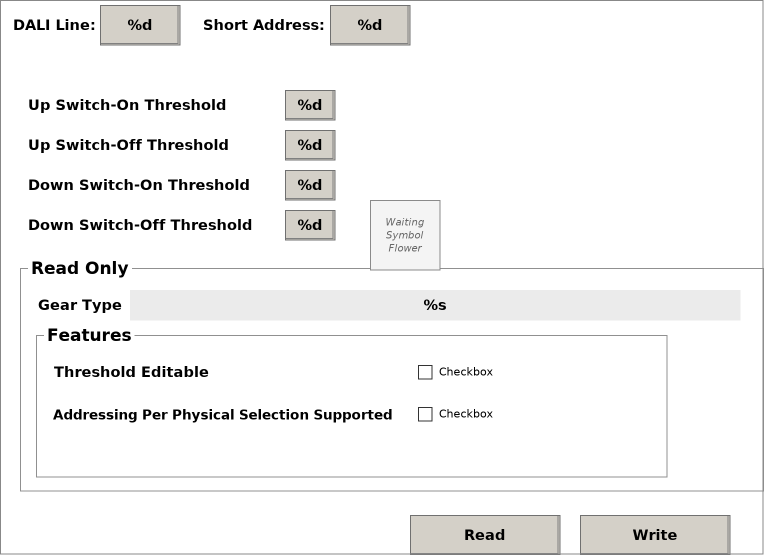
VISUALIZATION Visu_Part208Switching  // 764x555
    Group (200,5 210x40)
        Textfield (0,0 130x40), "Short Address:"
        Button (130,0 80x40), "%d", text variable: DALI_Commissioning.fbPart208Switching.nAddress
            OnMouseClick: write the text variable via Default, min 0, max 63, title "Insert Short Address"
    Group (10,5 170x40)
        Textfield (0,0 110x40), "DALI Line:"
        Button (90,0 80x40), "%d", text variable: GVL_Internal.nDALILine
            OnMouseClick: write the text variable via Default, min 1, max 10, title "Choose line"
    Textfield (25,90 250x30), "Up Switch-On Threshold"
    Textfield (25,130 250x30), "Up Switch-Off Threshold"
    Textfield (25,170 250x30), "Down Switch-On Threshold"
    Textfield (25,210 250x30), "Down Switch-Off Threshold"
    GroupBox (20,260 744x231), "Read Only"
        Textfield (15,30 250x30), "Gear Type"
        Textfield (110,30 610x30), "%s", text variable: DALI_Commissioning.fbPart208Switching.sGearType
        GroupBox (16,67 631x150), "Features"
            Checkbox (380,30 30x30), "Checkbox", variable: DALI_Commissioning.fbPart208Switching.bThreshold, input disabled if: TRUE
            Textfield (15,30 350x30), "Threshold Editable"
            Checkbox (380,72 30x30), "Checkbox", variable: DALI_Commissioning.fbPart208Switching.bAddressingPhysical, input disabled if: TRUE
    Textfield (50,400 355x30), "Addressing Per Physical Selection Supported"
    Button (410,515 150x40), "Read"
        OnMouseClick: execute { DALI_Commissioning.fbPart208Switching.bRead := TRUE; }
    Button (580,515 150x40), "Write"
        OnMouseClick: execute { DALI_Commissioning.fbPart208Switching.bWrite := TRUE; }
    WaitingSymbolFlower (370,200 70x70), invisible if: DALI_Commissioning.fbPart208Switching.bHideWaitSymbol
    Button (285,90 50x30), "%d", text variable: DALI_Commissioning.fbPart208Switching.nUpSwitchOnThreshold
        OnMouseClick: write the text variable via Default, min 0, max 255, title "Up Switch On Threshold"
    Button (285,130 50x30), "%d", text variable: DALI_Commissioning.fbPart208Switching.nUpSwitchOffThreshold
        OnMouseClick: write the text variable via Default, min 0, max 255, title "Up Switch Off Threshold"
    Button (285,170 50x30), "%d", text variable: DALI_Commissioning.fbPart208Switching.nDownSwitchOnThreshold
        OnMouseClick: write the text variable via Default, min 0, max 255, title "Down Switch On Threshold"
    Button (285,210 50x30), "%d", text variable: DALI_Commissioning.fbPart208Switching.nDownSwitchOffThreshold
        OnMouseClick: write the text variable via Default, min 0, max 255, title "Down Switch Off Threshold"
END_VISUALIZATION

(* stored: Version 1.1.0.1
   Visu Visu_Part208Switching: Id {15e6234d-45c9-48c5-8925-3509457e59ba} *)
